
FUNCTION CB_byte_to_int : INT

TITLE = ' Convert a byte into a Int '
VERSION : '1.0'
AUTHOR  : CB
NAME    : bytToInt
FAMILY  : TNI

VAR_INPUT
    IN : BYTE;
END_VAR

BEGIN

CB_byte_to_int := BYTE_TO_INT(IN);

END_FUNCTION
